// TIA Portal V19 export
VAR_GLOBAL   // PLC tag table "Equipment_Template_DefaultTagTable_4"
END_VAR
